% RSLogix 500 project Practica_6_Subrutinas.RSS, saved by version 8.30.00.16 %
PROJECT "UNTITLED"    % processor: MicroLogix 1000 %

PROGRAM FILES
  LAD 2 "MAIN_PROG"  8 rungs
  LAD 3 "USER_FAULT"  4 rungs
  LAD 4 "HSC_INT"  4 rungs
  LAD 5 "STI_INT"  1 rungs
  LAD 6, 7, 8, 9, 10, 11, 12, 13, 14, 15, 16: only END

DATA FILES
  O0 OUTPUT  1 elements
  I1 INPUT  2 elements
  S2 STATUS  33 elements
  B3 BINARY  32 elements
  T4 TIMER  40 elements
  C5 COUNTER  32 elements
  R6 CONTROL  16 elements
  N7 INTEGER  105 elements

LADDER 2 "MAIN_PROG"
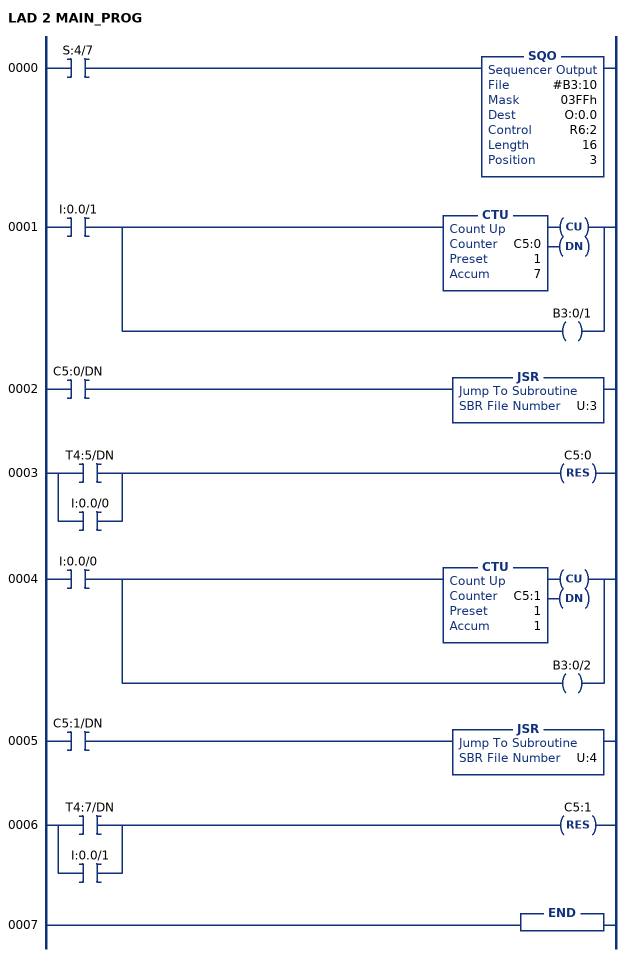
% Rung: 0 %
SOR XIC S:4/7 SQO #B3:10 03FFh O:0.0 R6:2 16 3 EOR
% Rung: 1 %
SOR XIC I:0.0/1 BST CTU C5:0 1 7 NXB OTE B3:0/1 BND EOR
% Rung: 2 %
SOR XIC C5:0/DN JSR U:3 EOR
% Rung: 3 %
SOR BST XIC T4:5/DN NXB XIC I:0.0/0 BND RES C5:0 EOR
% Rung: 4 %
SOR XIC I:0.0/0 BST CTU C5:1 1 1 NXB OTE B3:0/2 BND EOR
% Rung: 5 %
SOR XIC C5:1/DN JSR U:4 EOR
% Rung: 6 %
SOR BST XIC T4:7/DN NXB XIC I:0.0/1 BND RES C5:1 EOR
% Rung: 7 %
SOR END EOR

LADDER 3 "USER_FAULT"
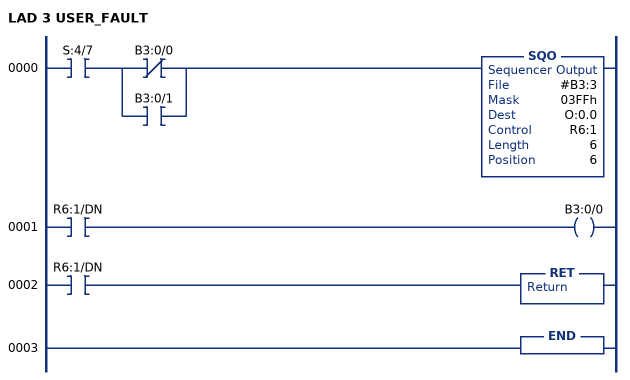
% Rung: 0 %
SOR XIC S:4/7 BST XIO B3:0/0 NXB XIC B3:0/1 BND SQO #B3:3 03FFh O:0.0 R6:1 6 6 EOR
% Rung: 1 %
SOR XIC R6:1/DN OTE B3:0/0 EOR
% Rung: 2 %
SOR XIC R6:1/DN RET EOR
% Rung: 3 %
SOR END EOR

LADDER 4 "HSC_INT"
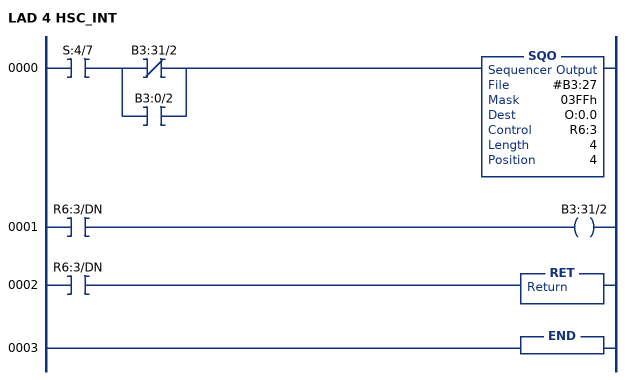
% Rung: 0 %
SOR XIC S:4/7 BST XIO B3:31/2 NXB XIC B3:0/2 BND SQO #B3:27 03FFh O:0.0 R6:3 4 4 EOR
% Rung: 1 %
SOR XIC R6:3/DN OTE B3:31/2 EOR
% Rung: 2 %
SOR XIC R6:3/DN RET EOR
% Rung: 3 %
SOR END EOR

OTHER DOCUMENTED ADDRESSES
  B3:10/0  "0"

REVISION NOTES
  0: ya con registros

DATA TABLE (non-zero values as saved)
DATA B3
% B3:0 % 0X0000 0X0000 0X0000 0X0000 0X0014 0X0014 0X0014 0X0012 0X0012 0X0012
% B3:10 % 0X0000 0X0041 0X0041 0X0001 0X0041 0X0001 0X0041 0X0021 0X0021 0X0014
% B3:20 % 0X0014 0X0010 0X0014 0X0010 0X0014 0X0012 0X0012 0X0000 0X0000 0X0041
% B3:30 % 0X0021 0X0004
DATA T4
% .PRE .ACC %
% T4:4 % 20 0
% T4:5 % 15 0
DATA C5
% .PRE .ACC %
% C5:0 % 1 7
% C5:1 % 1 1
DATA R6
% .LEN .POS %
% R6:1 % 6 6
% R6:2 % 16 3
% R6:3 % 4 4
